{region '#Template'}
	{attribute 'Version' := '5.0.0.0'}
	{attribute 'Tags' := '"LCID": "1031", "Text": "DUT, Enumeration, Betriebsart, Universal, 3Step"'}
	{attribute 'Tags' := '"LCID": "1033", "Text": "DUT, Enumeration, Operation mode, Universal, 3Step"'}
	{attribute 'Description' := '"LCID": "1031", "Text": "Betriebsart 3 3Step"'}
	{attribute 'Description' := '"LCID": "1033", "Text": "Operating mode 3 steps"'}
{endregion}

{attribute qualified_only}
TYPE E_BA_3Step :
(
	eOff			:= 1,
	eStep1			:= 2,
	eStep2			:= 3,
	eStep3			:= 4
	
) UDINT;
END_TYPE

(* stored: Version 1.1.0.1, ProductVersion 3.1.4024.12
   DUT E_BA_3Step: Id {8c606149-d03e-454b-958f-49d1843d27fe} *)
